// TIA Portal V16 export
// export: Created 2025-10-06T17:54:38.6495017Z, ExportSetting WithDefaults, DisplayName Totally Integrated Automation Portal, DisplayVersion V16, DisplayName TIA Portal Version Control Interface, DisplayVersion V16, DisplayName TIA Portal Openness, DisplayVersion V16, DisplayName STEP 7 Professional, DisplayVersion V16, DisplayName STEP 7 Safety, DisplayVersion V16, DisplayName WinCC Advanced, DisplayVersion V16
DATA_BLOCK "Delayed_Message_Function_Magazine"   // DB38
VERSION : 0.1
// stored: AutoNumber true, InstanceOfName Delayed_Message_Function, InstanceOfType FB
"Delayed_Message_Function"
   // VAR_INPUT
   //    "Override Message" : Bool;
   //    "Sensor Input 1" : Bool;
   //    "Sensor Input 2" : Bool;
   //    "Delay Time Message" : Time;
   //    "FlashTimer Time 1" : Time;
   //    "FlashTimer Time 2" : Time;
   // END_VAR
   // VAR_OUTPUT
   //    "Output Signal" : Bool;
   //    "Output Signal Halt" : Bool;
   //    "ET Delayed Timer" : Time;
   //    "Output LED Flashing" : Bool;
   // END_VAR
BEGIN
END_DATA_BLOCK
